// TIA Portal V17 export
// export: Created 2022-03-12T16:05:24.3318187Z, ExportSetting WithDefaults, DisplayName Totally Integrated Automation Portal, DisplayVersion V17, DisplayName TIA Portal Openness, DisplayVersion V17, DisplayName TIA Portal Version Control Interface, DisplayVersion V17, DisplayName STEP 7 Professional, DisplayVersion V17, DisplayName STEP 7 Safety, DisplayVersion V17, DisplayName WinCC Advanced / Unified PC, DisplayVersion V17
FUNCTION_BLOCK "EM02_00_Main"   // FB31680, LAD
TITLE = EM02_00_Main
{ S7_Optimized_Access := 'TRUE' }
AUTHOR : tech.team.motioncontrol@siemens.com
FAMILY : CPG
VERSION : 1.1
// Support: tech.team.motioncontrol@siemens.com
// stored: AutoNumber true, IsIECCheckEnabled false, IsRetainMemResEnabled false, MemoryReserve 100, SetENOAutomatically false, UDAEnableTagReadback false
   VAR
      instEventControl { ExternalAccessible := 'False'; ExternalVisible := 'False'; ExternalWritable := 'False'; S7_SetPoint := 'True'} : "EM02_01_EventControl";   // Instance DB - EM's Event Control Logic
      instPackML_ModuleSum { ExternalAccessible := 'False'; ExternalVisible := 'False'; ExternalWritable := 'False'; S7_SetPoint := 'True'} : "EM02_02_PackML_ModuleSum";   // Instance DB - EM's PackML Module Summation Logic
      instCM01 { ExternalAccessible := 'False'; ExternalVisible := 'False'; ExternalWritable := 'False'; S7_SetPoint := 'True'} : "EM02_CM01_Conveyor";   // Instance DB - CM01
      instCM02 { ExternalAccessible := 'False'; ExternalVisible := 'False'; ExternalWritable := 'False'; S7_SetPoint := 'True'} : "EM02_CM02_Palletizer";   // Instance DB - CM02
   END_VAR
   VAR_TEMP   // added for the SCL form of the ladder/FBD networks
      _w1 : Bool;
   END_VAR
BEGIN

REGION Network 1: *** BEGIN MAIN LOGIC SECTION ***
END_REGION

REGION Network 2: Call the Control Module Logic - CM01
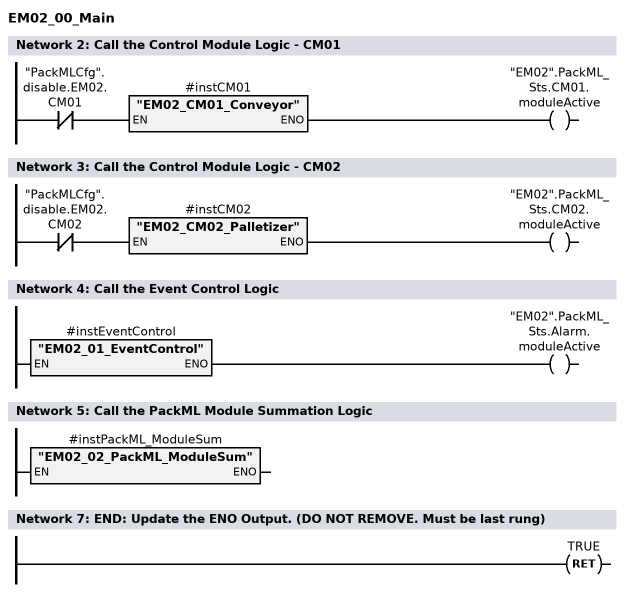
   RUNG wire#powerrail
      I_Contact( "PackMLCfg".disable.EM02.CM01 )
      #instCM01()
      Coil( "EM02".PackML_Sts.CM01.moduleActive )
   END_RUNG
   // the same network as SCL:
   #instCM01(EN := NOT "PackMLCfg".disable.EM02.CM01, ENO => #_w1);   // "EM02_CM01_Conveyor"
   "EM02".PackML_Sts.CM01.moduleActive := #_w1;
END_REGION

REGION Network 3: Call the Control Module Logic - CM02
   RUNG wire#powerrail
      I_Contact( "PackMLCfg".disable.EM02.CM02 )
      #instCM02()
      Coil( "EM02".PackML_Sts.CM02.moduleActive )
   END_RUNG
   // the same network as SCL:
   #instCM02(EN := NOT "PackMLCfg".disable.EM02.CM02, ENO => #_w1);   // "EM02_CM02_Palletizer"
   "EM02".PackML_Sts.CM02.moduleActive := #_w1;
END_REGION

REGION Network 4: Call the Event Control Logic
   RUNG wire#powerrail
      #instEventControl()
      Coil( "EM02".PackML_Sts.Alarm.moduleActive )
   END_RUNG
   // the same network as SCL:
   #instEventControl(ENO => #_w1);   // "EM02_01_EventControl"
   "EM02".PackML_Sts.Alarm.moduleActive := #_w1;
END_REGION

REGION Network 5: Call the PackML Module Summation Logic
   RUNG wire#powerrail
      #instPackML_ModuleSum()
   END_RUNG
   // the same network as SCL:
   #instPackML_ModuleSum();   // "EM02_02_PackML_ModuleSum"
END_REGION

REGION Network 7: END: Update the ENO Output. (DO NOT REMOVE. Must be last rung)
   RUNG wire#powerrail
      ReturnCoil( TRUE )
   END_RUNG
   // the same network as SCL:
   ENO := TRUE;
   RETURN;
END_REGION
END_FUNCTION_BLOCK
